{attribute 'linkalways'} 
{attribute 'no_explicit_call' := 'This FB is a CLASS and must be accessed using methods or properties'}
{attribute 'enable_dynamic_creation'}
FUNCTION_BLOCK Node_F_VN_ContourEccentricity EXTENDS VisionNode
VAR
    ipContour : _ITcVnContainer;
    fEccentricity : _LREAL(0.0);
    hrPrev : _HRESULT(S_OK);
	hresult : _HRESULT(S_OK);
END_VAR

METHOD PUBLIC  Clone : I_Node
VAR
	pNode : POINTER TO Node_F_VN_ContourEccentricity;
END_VAR
pNode := __NEW(Node_F_VN_ContourEccentricity);
Clone := pNode^;
END_METHOD

METHOD FB_init : BOOL
VAR_INPUT
	bInitRetains : BOOL; // if TRUE, the retain variables are initialized (warm start / cold start)
	bInCopyCode : BOOL;  // if TRUE, the instance afterwards gets moved into the copy code (online change)
END_VAR
AddInput('ipContour', ipContour);
AddInput('hrPrev', hrPrev);
AddOutput('fEccentricity', fEccentricity);
AddOutput('hresult',hresult);
END_METHOD

METHOD PROTECTED OnExecute
hresult.Value := F_VN_ContourEccentricity(
	ipContour := ipContour.Value,
    fEccentricity := fEccentricity.Value,
	hrPrev:= hrPrev.Value);
END_METHOD

METHOD PUBLIC PreExecutionCheck
VAR_INPUT
	Check : I_PreExecutionChecks;
END_VAR
Check.IsTrue(ipContour.IsValid, 'ipContour must be a valid container');
Check.IsTrue((ipContour.IsType(TC_GLOBAL_CONST_LIST.ContainerType_Vector_TcVnPoint2_DINT) OR
              ipContour.IsType(TC_GLOBAL_CONST_LIST.ContainerType_Vector_TcVnPoint2_REAL)),
              'ipContour contains incorrect type');
END_METHOD

END_FUNCTION_BLOCK

(* stored: Version 1.1.0.1, ProductVersion 3.1.4026.13
   POU Node_F_VN_ContourEccentricity: Id {3b4d1af3-83a3-0ccf-0fdc-24605fbce745}, SpecialFunc None
   Folder Constructor: Id {c9a337ad-5c12-05bb-0858-8090dac10b56}
   Method Clone: Id {b5b7d43e-9452-07b5-2f0d-4767fee70370}
   Method FB_init: Id {54879b11-a17c-0298-0262-528df0f33fa7}
   Method OnExecute: Id {481c0427-da59-0974-20c5-78a415f60ad4}
   Method PreExecutionCheck: Id {42afe8ba-0e81-06d4-1dcb-490e00fb8d3d} *)
